// TIA Portal V17 export
// export: Created 2026-04-13T11:12:52.9655519Z, ExportSetting WithDefaults, DisplayName Totally Integrated Automation Portal, DisplayVersion V17 Update 4, DisplayName TIA Portal Openness, DisplayVersion V17 Update 4, DisplayName TIA Portal Version Control Interface, DisplayVersion V17, DisplayName SINAMICS Startdrive Advanced, DisplayVersion V17, DisplayName SINAMICS Startdrive G130, G150, S120, S150, SINAMICS MV, S210, DisplayVersion V17, DisplayName SINAMICS Startdrive G110M, G120, G120C, G120D, G120P, G115D, DisplayVersion V17, DisplayName STEP 7 Professional, DisplayVersion V17 Update 4, DisplayName STEP 7 Safety, DisplayVersion V17, DisplayName WinCC Professional, DisplayVersion V17 Update 4
TagTable "IOM"
  IBD补氮阀关反馈 : Bool  (PLC tag IBD补氮阀关反馈, HMI_连接_1, 1 s)
  IBD补氮阀开反馈 : Bool  (PLC tag IBD补氮阀开反馈, HMI_连接_1, 1 s)
  IBP爆破片1反馈 : Bool  (PLC tag IBP爆破片1反馈, HMI_连接_1, 1 s)
  IBP爆破片2反馈 : Bool  (PLC tag IBP爆破片2反馈, HMI_连接_1, 1 s)
  IBS闭式进风隔断阀关反馈 : Bool  (PLC tag IBS闭式进风隔断阀关反馈, HMI_连接_1, 1 s)
  IBS闭式进风隔断阀开反馈 : Bool  (PLC tag IBS闭式进风隔断阀开反馈, HMI_连接_1, 1 s)
  IBS闭式排风隔断阀关反馈 : Bool  (PLC tag IBS闭式排风隔断阀关反馈, HMI_连接_1, 1 s)
  IBS闭式排风隔断阀开反馈 : Bool  (PLC tag IBS闭式排风隔断阀开反馈, HMI_连接_1, 1 s)
  ICW除雾排液阀关反馈 : Bool  (PLC tag ICW除雾排液阀关反馈, HMI_连接_1, 1 s)
  ICW除雾排液阀开反馈 : Bool  (PLC tag ICW除雾排液阀开反馈, HMI_连接_1, 1 s)
  IDJ电加热 : Bool  (PLC tag IDJ电加热, HMI_连接_1, 1 s)
  IEJ二级冷冻水阀关反馈 : Bool  (PLC tag IEJ二级冷冻水阀关反馈, HMI_连接_1, 1 s)
  IEJ二级冷冻水阀开反馈 : Bool  (PLC tag IEJ二级冷冻水阀开反馈, HMI_连接_1, 1 s)
  IEJ二级排液阀关反馈 : Bool  (PLC tag IEJ二级排液阀关反馈, HMI_连接_1, 1 s)
  IEJ二级排液阀开反馈 : Bool  (PLC tag IEJ二级排液阀开反馈, HMI_连接_1, 1 s)
  IJD进氮阀关反馈 : Bool  (PLC tag IJD进氮阀关反馈, HMI_连接_1, 1 s)
  IJD进氮阀开反馈 : Bool  (PLC tag IJD进氮阀开反馈, HMI_连接_1, 1 s)
  IJF进风保护温度 : Bool  (PLC tag IJF进风保护温度, HMI_连接_1, 1 s)
  IJF进风冷却水阀关反馈 : Bool  (PLC tag IJF进风冷却水阀关反馈, HMI_连接_1, 1 s)
  IJF进风冷却水阀开反馈 : Bool  (PLC tag IJF进风冷却水阀开反馈, HMI_连接_1, 1 s)
  IJF进风冷却水流量 : Bool  (PLC tag IJF进风冷却水流量, HMI_连接_1, 1 s)
  IJL进料泵 : Bool  (PLC tag IJL进料泵, HMI_连接_1, 1 s)
  IJT急停 : Bool  (PLC tag IJT急停, HMI_连接_1, 1 s)
  IKS开式进风隔断阀关反馈 : Bool  (PLC tag IKS开式进风隔断阀关反馈, HMI_连接_1, 1 s)
  IKS开式进风隔断阀开反馈 : Bool  (PLC tag IKS开式进风隔断阀开反馈, HMI_连接_1, 1 s)
  IKS开式排风隔断阀关反馈 : Bool  (PLC tag IKS开式排风隔断阀关反馈, HMI_连接_1, 1 s)
  IKS开式排风隔断阀开反馈 : Bool  (PLC tag IKS开式排风隔断阀开反馈, HMI_连接_1, 1 s)
  ILD冷冻水流量 : Bool  (PLC tag ILD冷冻水流量, HMI_连接_1, 1 s)
  ILQ冷却水流量 : Bool  (PLC tag ILQ冷却水流量, HMI_连接_1, 1 s)
  ILX离心雾化器 : Bool  (PLC tag ILX离心雾化器, HMI_连接_1, 1 s)
  IPY排液流量 : Bool  (PLC tag IPY排液流量, HMI_连接_1, 1 s)
  IQL气流雾化阀关反馈 : Bool  (PLC tag IQL气流雾化阀关反馈, HMI_连接_1, 1 s)
  IQL气流雾化阀开反馈 : Bool  (PLC tag IQL气流雾化阀开反馈, HMI_连接_1, 1 s)
  IQX清洗伸缩气缸降反馈 : Bool  (PLC tag IQX清洗伸缩气缸降反馈, HMI_连接_1, 1 s)
  IQX清洗伸缩气缸升反馈 : Bool  (PLC tag IQX清洗伸缩气缸升反馈, HMI_连接_1, 1 s)
  IRJ溶剂回收排放阀关反馈 : Bool  (PLC tag IRJ溶剂回收排放阀关反馈, HMI_连接_1, 1 s)
  IRJ溶剂回收排放阀开反馈 : Bool  (PLC tag IRJ溶剂回收排放阀开反馈, HMI_连接_1, 1 s)
  IRJ溶剂排液泵关反馈 : Bool  (PLC tag IRJ溶剂排液泵关反馈, HMI_连接_1, 1 s)
  IRJ溶剂排液泵开反馈 : Bool  (PLC tag IRJ溶剂排液泵开反馈, HMI_连接_1, 1 s)
  ISF输送风机 : Bool  (PLC tag ISF输送风机, HMI_连接_1, 1 s)
  ISF输送加热 : Bool  (PLC tag ISF输送加热, HMI_连接_1, 1 s)
  ISF输送进风阀关反馈 : Bool  (PLC tag ISF输送进风阀关反馈, HMI_连接_1, 1 s)
  ISF输送进风阀开反馈 : Bool  (PLC tag ISF输送进风阀开反馈, HMI_连接_1, 1 s)
  ISF送风机 : Bool  (PLC tag ISF送风机, HMI_连接_1, 1 s)
  ISN室内排水关反馈 : Bool  (PLC tag ISN室内排水关反馈, HMI_连接_1, 1 s)
  ISN室内排水开反馈 : Bool  (PLC tag ISN室内排水开反馈, HMI_连接_1, 1 s)
  ISS输送保护温度 : Bool  (PLC tag ISS输送保护温度, HMI_连接_1, 1 s)
  ITD塔顶清洗球阀关反馈 : Bool  (PLC tag ITD塔顶清洗球阀关反馈, HMI_连接_1, 1 s)
  ITD塔顶清洗球阀开反馈 : Bool  (PLC tag ITD塔顶清洗球阀开反馈, HMI_连接_1, 1 s)
  IXY泄压阀关反馈 : Bool  (PLC tag IXY泄压阀关反馈, HMI_连接_1, 1 s)
  IXY泄压阀开反馈 : Bool  (PLC tag IXY泄压阀开反馈, HMI_连接_1, 1 s)
  IYF引风机 : Bool  (PLC tag IYF引风机, HMI_连接_1, 1 s)
  IYJ一级冷却水阀关反馈 : Bool  (PLC tag IYJ一级冷却水阀关反馈, HMI_连接_1, 1 s)
  IYJ一级冷却水阀开反馈 : Bool  (PLC tag IYJ一级冷却水阀开反馈, HMI_连接_1, 1 s)
  IYJ一级排液阀关反馈 : Bool  (PLC tag IYJ一级排液阀关反馈, HMI_连接_1, 1 s)
  IYJ一级排液阀开反馈 : Bool  (PLC tag IYJ一级排液阀开反馈, HMI_连接_1, 1 s)
  QASA室内回水阀 : Bool  (PLC tag QASA室内回水阀, HMI_连接_1, 1 s)
  QASA室外回水阀 : Bool  (PLC tag QASA室外回水阀, HMI_连接_1, 1 s)
  QBD补氮阀 : Bool  (PLC tag QBD补氮阀, HMI_连接_1, 1 s)
  QBD布袋振打1 : Bool  (PLC tag QBD布袋振打1, HMI_连接_1, 1 s)
  QBD布袋振打3 : Bool  (PLC tag QBD布袋振打3, HMI_连接_1, 1 s)
  QBD布袋振打4 : Bool  (PLC tag QBD布袋振打4, HMI_连接_1, 1 s)
  QBS闭式进风隔断阀 : Bool  (PLC tag QBS闭式进风隔断阀, HMI_连接_1, 1 s)
  QBS闭式排风隔断阀 : Bool  (PLC tag QBS闭式排风隔断阀, HMI_连接_1, 1 s)
  QBY备用1 : Bool  (PLC tag QBY备用1, HMI_连接_1, 1 s)
  QBY备用2 : Bool  (PLC tag QBY备用2, HMI_连接_1, 1 s)
  QBY备用3 : Bool  (PLC tag QBY备用3, HMI_连接_1, 1 s)
  QBY备用4 : Bool  (PLC tag QBY备用4, HMI_连接_1, 1 s)
  QBY备用7 : Bool  (PLC tag QBY备用7, HMI_连接_1, 1 s)
  QBY备用10 : Bool  (PLC tag QBY备用10, HMI_连接_1, 1 s)
  QBY备用11 : Bool  (PLC tag QBY备用11, HMI_连接_1, 1 s)
  QBY备用12 : Bool  (PLC tag QBY备用12, HMI_连接_1, 1 s)
  QBY备用13 : Bool  (PLC tag QBY备用13, HMI_连接_1, 1 s)
  QBY备用14 : Bool  (PLC tag QBY备用14, HMI_连接_1, 1 s)
  QBY备用15 : Bool  (PLC tag QBY备用15, HMI_连接_1, 1 s)
  QBY备用16 : Bool  (PLC tag QBY备用16, HMI_连接_1, 1 s)
  QBY备用17 : Bool  (PLC tag QBY备用17, HMI_连接_1, 1 s)
  QBY备用18 : Bool  (PLC tag QBY备用18, HMI_连接_1, 1 s)
  QBY备用19 : Bool  (PLC tag QBY备用19, HMI_连接_1, 1 s)
  QBY备用20 : Bool  (PLC tag QBY备用20, HMI_连接_1, 1 s)
  QCC除尘出料上阀 : Bool  (PLC tag QCC除尘出料上阀, HMI_连接_1, 1 s)
  QCC除尘出料下阀 : Bool  (PLC tag QCC除尘出料下阀, HMI_连接_1, 1 s)
  QCC除尘管道清洗阀 : Bool  (PLC tag QCC除尘管道清洗阀, HMI_连接_1, 1 s)
  QCC除尘缓存震荡器 : Bool  (PLC tag QCC除尘缓存震荡器, HMI_连接_1, 1 s)
  QCC除尘脉冲 : Bool  (PLC tag QCC除尘脉冲, HMI_连接_1, 1 s)
  QCC除尘气锤1 : Bool  (PLC tag QCC除尘气锤1, HMI_连接_1, 1 s)
  QCC除尘气锤2 : Bool  (PLC tag QCC除尘气锤2, HMI_连接_1, 1 s)
  QCC除尘清洗阀 : Bool  (PLC tag QCC除尘清洗阀, HMI_连接_1, 1 s)
  QCF出风高效清洗阀 : Bool  (PLC tag QCF出风高效清洗阀, HMI_连接_1, 1 s)
  QCIP启动 : Bool  (PLC tag QCIP启动, HMI_连接_1, 1 s)
  QCS纯水洗请求 : Bool  (PLC tag QCS纯水洗请求, HMI_连接_1, 1 s)
  QCW除雾排液阀 : Bool  (PLC tag QCW除雾排液阀, HMI_连接_1, 1 s)
  QDJ电加热器 : Bool  (PLC tag QDJ电加热器, HMI_连接_1, 1 s)
  QEJ二级出料上阀 : Bool  (PLC tag QEJ二级出料上阀, HMI_连接_1, 1 s)
  QEJ二级出料下阀 : Bool  (PLC tag QEJ二级出料下阀, HMI_连接_1, 1 s)
  QEJ二级缓存震荡器 : Bool  (PLC tag QEJ二级缓存震荡器, HMI_连接_1, 1 s)
  QEJ二级冷冻水阀 : Bool  (PLC tag QEJ二级冷冻水阀, HMI_连接_1, 1 s)
  QEJ二级冷凝清洗阀 : Bool  (PLC tag QEJ二级冷凝清洗阀, HMI_连接_1, 1 s)
  QEJ二级排液阀 : Bool  (PLC tag QEJ二级排液阀, HMI_连接_1, 1 s)
  QEJ二级旋风清洗阀 : Bool  (PLC tag QEJ二级旋风清洗阀, HMI_连接_1, 1 s)
  QEJ二级旋风振打锤 : Bool  (PLC tag QEJ二级旋风振打锤, HMI_连接_1, 1 s)
  QFM蜂鸣器 : Bool  (PLC tag QFM蜂鸣器, HMI_连接_1, 1 s)
  QGS供水泵启动 : Bool  (PLC tag QGS供水泵启动, HMI_连接_1, 1 s)
  QHF回风蒸汽开关阀 : Bool  (PLC tag QHF回风蒸汽开关阀, HMI_连接_1, 1 s)
  QHF回风蒸汽排水阀 : Bool  (PLC tag QHF回风蒸汽排水阀, HMI_连接_1, 1 s)
  QHF回风蒸汽调节阀 : Bool  (PLC tag QHF回风蒸汽调节阀, HMI_连接_1, 1 s)
  QHS回水隔断阀1 : Bool  (PLC tag QHS回水隔断阀1, HMI_连接_1, 1 s)
  QJD进氮阀 : Bool  (PLC tag QJD进氮阀, HMI_连接_1, 1 s)
  QJF进风冷却水阀 : Bool  (PLC tag QJF进风冷却水阀, HMI_连接_1, 1 s)
  QJF进风蒸汽比例调节阀 : Bool  (PLC tag QJF进风蒸汽比例调节阀, HMI_连接_1, 1 s)
  QJF进风蒸汽开关阀 : Bool  (PLC tag QJF进风蒸汽开关阀, HMI_连接_1, 1 s)
  QJF进风蒸汽排水阀 : Bool  (PLC tag QJF进风蒸汽排水阀, HMI_连接_1, 1 s)
  QJL进料泵 : Bool  (PLC tag QJL进料泵, HMI_连接_1, 1 s)
  QJL进料泵风扇 : Bool  (PLC tag QJL进料泵风扇, HMI_连接_1, 1 s)
  QJR加热清洗阀 : Bool  (PLC tag QJR加热清洗阀, HMI_连接_1, 1 s)
  QJS碱水洗请求 : Bool  (PLC tag QJS碱水洗请求, HMI_连接_1, 1 s)
  QKS开式进风隔断阀 : Bool  (PLC tag QKS开式进风隔断阀, HMI_连接_1, 1 s)
  QKS开式排风隔断阀 : Bool  (PLC tag QKS开式排风隔断阀, HMI_连接_1, 1 s)
  QLC料仓清洗阀 : Bool  (PLC tag QLC料仓清洗阀, HMI_连接_1, 1 s)
  QLC料仓清洗排水阀 : Bool  (PLC tag QLC料仓清洗排水阀, HMI_连接_1, 1 s)
  QLG料罐清洗阀 : Bool  (PLC tag QLG料罐清洗阀, HMI_连接_1, 1 s)
  QLX离心雾化 : Bool  (PLC tag QLX离心雾化, HMI_连接_1, 1 s)
  QLX离心雾化风扇 : Bool  (PLC tag QLX离心雾化风扇, HMI_连接_1, 1 s)
  QLX离心雾化油泵 : Bool  (PLC tag QLX离心雾化油泵, HMI_连接_1, 1 s)
  QPH平衡比例调节阀 : Bool  (PLC tag QPH平衡比例调节阀, HMI_连接_1, 1 s)
  QQG气缸降 : Bool  (PLC tag QQG气缸降, HMI_连接_1, 1 s)
  QQG气缸升 : Bool  (PLC tag QQG气缸升, HMI_连接_1, 1 s)
  QQG气缸升降阀 : Bool  (PLC tag QQG气缸升降阀, HMI_连接_1, 1 s)
  QQL气流雾化阀 : Bool  (PLC tag QQL气流雾化阀, HMI_连接_1, 1 s)
  QQS缺水状态 : Bool  (PLC tag QQS缺水状态, HMI_连接_1, 1 s)
  QQX清洗溶剂出阀 : Bool  (PLC tag QQX清洗溶剂出阀, HMI_连接_1, 1 s)
  QQZ前置水阀 : Bool  (PLC tag QQZ前置水阀, HMI_连接_1, 1 s)
  QRC热纯自动洗 : Bool  (PLC tag QRC热纯自动洗, HMI_连接_1, 1 s)
  QRJ溶剂回收排放阀 : Bool  (PLC tag QRJ溶剂回收排放阀, HMI_连接_1, 1 s)
  QRJ溶剂进程泵 : Bool  (PLC tag QRJ溶剂进程泵, HMI_连接_1, 1 s)
  QRJ溶剂排液泵 : Bool  (PLC tag QRJ溶剂排液泵, HMI_连接_1, 1 s)
  QRJ溶剂排液泵进阀 : Bool  (PLC tag QRJ溶剂排液泵进阀, HMI_连接_1, 1 s)
  QRJ溶剂请求 : Bool  (PLC tag QRJ溶剂请求, HMI_连接_1, 1 s)
  QRJ溶剂洗 : Bool  (PLC tag QRJ溶剂洗, HMI_连接_1, 1 s)
  QRS热水洗请求 : Bool  (PLC tag QRS热水洗请求, HMI_连接_1, 1 s)
  QSB设备振打 : Bool  (PLC tag QSB设备振打, HMI_连接_1, 1 s)
  QSF送风机 : Bool  (PLC tag QSF送风机, HMI_连接_1, 1 s)
  QSF送风机风扇 : Bool  (PLC tag QSF送风机风扇, HMI_连接_1, 1 s)
  QSF送风机排水阀 : Bool  (PLC tag QSF送风机排水阀, HMI_连接_1, 1 s)
  QSF送风机清洗阀 : Bool  (PLC tag QSF送风机清洗阀, HMI_连接_1, 1 s)
  QSJ水进程泵 : Bool  (PLC tag QSJ水进程泵, HMI_连接_1, 1 s)
  QSN室内排水隔膜泵 : Bool  (PLC tag QSN室内排水隔膜泵, HMI_连接_1, 1 s)
  QSN室内清洗总阀 : Bool  (PLC tag QSN室内清洗总阀, HMI_连接_1, 1 s)
  QSS输送出料上阀 : Bool  (PLC tag QSS输送出料上阀, HMI_连接_1, 1 s)
  QSS输送出料下阀 : Bool  (PLC tag QSS输送出料下阀, HMI_连接_1, 1 s)
  QSS输送风机 : Bool  (PLC tag QSS输送风机, HMI_连接_1, 1 s)
  QSS输送管路排水阀 : Bool  (PLC tag QSS输送管路排水阀, HMI_连接_1, 1 s)
  QSS输送管路清洗阀 : Bool  (PLC tag QSS输送管路清洗阀, HMI_连接_1, 1 s)
  QSS输送加热器 : Bool  (PLC tag QSS输送加热器, HMI_连接_1, 1 s)
  QSS输送进风阀 : Bool  (PLC tag QSS输送进风阀, HMI_连接_1, 1 s)
  QTD塔顶清洗球阀 : Bool  (PLC tag QTD塔顶清洗球阀, HMI_连接_1, 1 s)
  QWK蜗壳清洗阀 : Bool  (PLC tag QWK蜗壳清洗阀, HMI_连接_1, 1 s)
  QWL物料进阀 : Bool  (PLC tag QWL物料进阀, HMI_连接_1, 1 s)
  QXF旋风管道清洗阀 : Bool  (PLC tag QXF旋风管道清洗阀, HMI_连接_1, 1 s)
  QXT心跳发送信号 : Bool  (PLC tag QXT心跳发送信号, HMI_连接_1, 100 ms)
  QXY泄压阀 : Bool  (PLC tag QXY泄压阀, HMI_连接_1, 1 s)
  QYF引风机 : Bool  (PLC tag QYF引风机, HMI_连接_1, 1 s)
  QYF引风机风扇 : Bool  (PLC tag QYF引风机风扇, HMI_连接_1, 1 s)
  QYF引风机排水阀 : Bool  (PLC tag QYF引风机排水阀, HMI_连接_1, 1 s)
  QYF引风机清洗阀 : Bool  (PLC tag QYF引风机清洗阀, HMI_连接_1, 1 s)
  QYG压干请求 : Bool  (PLC tag QYG压干请求, HMI_连接_1, 1 s)
  QYH氧含仪隔断阀 : Bool  (PLC tag QYH氧含仪隔断阀, HMI_连接_1, 1 s)
  QYJ一级出料上阀 : Bool  (PLC tag QYJ一级出料上阀, HMI_连接_1, 1 s)
  QYJ一级出料下阀 : Bool  (PLC tag QYJ一级出料下阀, HMI_连接_1, 1 s)
  QYJ一级缓存振荡器 : Bool  (PLC tag QYJ一级缓存振荡器, HMI_连接_1, 1 s)
  QYJ一级冷凝清洗阀 : Bool  (PLC tag QYJ一级冷凝清洗阀, HMI_连接_1, 1 s)
  QYJ一级冷却水阀 : Bool  (PLC tag QYJ一级冷却水阀, HMI_连接_1, 1 s)
  QYJ一级排液阀 : Bool  (PLC tag QYJ一级排液阀, HMI_连接_1, 1 s)
  QYJ一级旋风清洗阀 : Bool  (PLC tag QYJ一级旋风清洗阀, HMI_连接_1, 1 s)
  QYJ一级旋风振打锤 : Bool  (PLC tag QYJ一级旋风振打锤, HMI_连接_1, 1 s)
  QYJ一级旋风振荡器 : Bool  (PLC tag QYJ一级旋风振荡器, HMI_连接_1, 1 s)
  QYS钥匙开关 : Bool  (PLC tag QYS钥匙开关, HMI_连接_1, 1 s)
  QZM照明灯 : Bool  (PLC tag QZM照明灯, HMI_连接_1, 1 s)
  QZS指示灯 : Bool  (PLC tag QZS指示灯, HMI_连接_1, 1 s)
  QZS注射水洗 : Bool  (PLC tag QZS注射水洗, HMI_连接_1, 1 s)
  QZT主塔排水阀 : Bool  (PLC tag QZT主塔排水阀, HMI_连接_1, 1 s)
  QZT主塔气锤1 : Bool  (PLC tag QZT主塔气锤1, HMI_连接_1, 1 s)
  QZT主塔气锤2 : Bool  (PLC tag QZT主塔气锤2, HMI_连接_1, 1 s)
  QZT主塔气锤3 : Bool  (PLC tag QZT主塔气锤3, HMI_连接_1, 1 s)
  QZT主塔气锤4 : Bool  (PLC tag QZT主塔气锤4, HMI_连接_1, 1 s)
  QZT主塔清洗进水阀 : Bool  (PLC tag QZT主塔清洗进水阀, HMI_连接_1, 100 ms)
